// TIA Portal V16 export
// export: Created 2021-05-25T16:14:39.4449537Z, ExportSetting WithDefaults, DisplayName Totally Integrated Automation Portal, DisplayVersion V16, DisplayName TIA Portal Version Control Interface, DisplayVersion V16, DisplayName TIA Portal Openness, DisplayVersion V16, DisplayName STEP 7 Professional, DisplayVersion V16, DisplayName STEP 7 Safety, DisplayVersion V16, DisplayName WinCC Unified SCADA Engineering System, DisplayVersion V16
DATA_BLOCK "dbHMIUser"   // DB5
{ S7_Optimized_Access := 'FALSE'; DB_Accessible_From_OPC_UA := 'FALSE' }
VERSION : 0.1
// stored: AutoNumber false, DBAccessibleFromOPCUA false, IsOnlyStoredInLoadMemory false, IsWriteProtectedInAS false
   VAR
      CurrentUsername : String;
      Spare_Bool0 : Bool;
      Spare_2 : Int;
      Spare_3 : Int;
      Spare_4 : UDInt;
      Spare_5 : UDInt;
      Spare_1 : Int;
      SetTargetHMIScreen : Byte;
      HMIScreenJobNo_byte1 : Byte;
      HMIScreenJobNo_byte2 : Byte;
      HMIScreenJobNo_byte3 : Byte;
      HMICurrScreen : Byte;
      HMIScreenJobNo_byte5 : Byte;
      HMIScreenJobNo_byte6 : Byte;
      HMIScreenJobNo_byte7 : Byte;
      HMIScreenJobNo_byte8 : Byte;
      HMIScreenJobNo_byte9 : Byte;
      HMIScreenJobNo_byte10 : Byte;
      HMIScreenJobNo_byte11 : Byte;
      HMIScreenJobNo_byte12 : Byte;
      HMIScreenJobNo_byte13 : Byte;
      HMIScreenJobNo_byte14 : Byte;
      HMIScreenJobNo_byte15 : Byte;
      HMIScreenJobNo_byte16 : Byte;
      HMIScreenJobNo_byte17 : Byte;
      Spare_6 : Int;
      PLCUserLogOut : Int;
      CurrUser_LEN : Int;
      UserLoggOffTime : UDInt := 50;
      CurrMachineStep : String[50];
      HMICurrScreen_OLD { ExternalAccessible := 'False'; ExternalVisible := 'False'; ExternalWritable := 'False'} : Byte;
      PLCUserLogOut_OLD { ExternalAccessible := 'False'; ExternalVisible := 'False'; ExternalWritable := 'False'} : Int;
   END_VAR
BEGIN
END_DATA_BLOCK
